{attribute addProperty BoxType "EL4732-0001-0000"}
{attribute addProperty Id "Value1AT %Q*INT1621Value2AT %Q*INT1621"}
{attribute addProperty CRC "1840860122"}
{attribute addProperty SizeInBites "32"}
{attribute addProperty SizeInBytes "4"}
TYPE Sample_6DB94BDA :
STRUCT
	{attribute addProperty Name "Value1"}
	Value1 AT %Q* : INT;
	{attribute addProperty Name "Value2"}
	Value2 AT %Q* : INT;
END_STRUCT
END_TYPE

(* stored: Version 1.2.0.0, ProductVersion 3.1.4024.9
   DUT Sample_6DB94BDA: Id {759f2932-3893-4c5f-ad44-65de1c4880e6} *)
